//Used to register fast faults
FUNCTION_BLOCK FB_UsualSuspects
VAR_INPUT
	
END_VAR
VAR_OUTPUT
	
END_VAR
VAR
	asList	:	ARRAY[0..99] OF T_MaxString;
	fbListController	:	FB_StringRingBuffer :=(
		bOverwrite := FALSE); //Throw error if list is full
END_VAR

METHOD M_Register : BOOL
VAR_INPUT
	i_sFFName	:	STRING; //Fast fault FB variable name to register
END_VAR

THIS^.fbListController.A_AddTail(
	putValue := i_sFFName,
	pBuffer	:=	ADR(THIS^.asList),
	cbBuffer	:=	SIZEOF(THIS^.asList),
	bOverwrite := FALSE);
	
M_Register := THIS^.fbListController.bOk; //TRUE if add succeeded
END_METHOD

END_FUNCTION_BLOCK

(* stored: Version 1.1.0.1, ProductVersion 3.1.4022.18
   POU FB_UsualSuspects: Id {b6e8568a-ba54-05c5-19d2-5d73b81187c6}, SpecialFunc None
   Method M_Register: Id {8c330f28-6df8-02bf-16cf-e775a52233cb} *)
